// TwinCAT 3 PLC project PLC1
// ProgramVersion: 3.1.4024.12
// libraries:
//   SG_Servo, * (SG)
//   Tc2_Standard, * (Beckhoff Automation GmbH)
//   Tc2_System, * (Beckhoff Automation GmbH)
//   Tc3_Module, * (Beckhoff Automation GmbH)
// project tree:
//   / PlcTask.TcTTO
//   POUs/ MAIN.TcPOU, DeviceState.TcPOU, UN01.TcPOU
// real-time tasks:
//   TASK PlcTask: cycle T#1ms, priority 20, ADS port 350
// motion (NC):
//   TASK NC-Task 1 SAF: cycle T#2ms, priority 4, ADS port 501
//   TASK NC-Task 1 SVB: cycle T#10ms, priority 8, ADS port 511
//   AXIS EM04-M1 (id 1)
//     Dynamic: AccelerationMaximum=2000, DecelerationMaximum=2000, Acceleration=926.842, Deceleration=926.842, Jerk=2000
//     Velo: RefSearch=6.17895, RefSync=6.17895, SlowManual=50, FastManual=200, Fast=617.895, Maximum=200
//     OtherSettings: AllowMotionCmdToSlave=true
//     encoder EncType=19
//       EncPara: ScaleFactorNumerator=12560, ScaleFactorDenominator=1907359744, Inverse=true, MaxCount=#xffffffff
//     drive DrvType=16
//       DrvPara: Inverse=true, MaxCount=#xffffffff, DriveControlDWord=#x00020000
//         Analog: VeloReferenz=679.6845, VeloScale=32, TorqueSetpointScale=10, ScaleFactorActTorque=0.1
//         TimeComp: TaskDelayCycles=1
//     controller CtrType=1
//       CtrPara: PriorControlFactor=1
//         Observer: BandWidth=20
//   AXIS EM05-M1 (id 2)
//     Dynamic: AccelerationMaximum=2000, DecelerationMaximum=2000, Acceleration=926.842, Deceleration=926.842, Jerk=2000
//     Velo: RefSearch=6.17895, RefSync=6.17895, SlowManual=50, FastManual=200, Fast=617.895, Maximum=200
//     OtherSettings: AllowMotionCmdToSlave=true
//     encoder EncType=19
//       EncPara: ScaleFactorNumerator=12560, ScaleFactorDenominator=1907359744, MaxCount=#xffffffff
//     drive DrvType=16
//       DrvPara: MaxCount=#xffffffff, DriveControlDWord=#x00020000
//         Analog: VeloReferenz=679.6845, VeloScale=32, TorqueSetpointScale=10, ScaleFactorActTorque=0.1
//         TimeComp: TaskDelayCycles=1
//     controller CtrType=1
//       CtrPara: PriorControlFactor=1
//         Observer: BandWidth=20
//   AXIS EM07-M1 (id 3)
//     Dynamic: AccelerationMaximum=1000, DecelerationMaximum=1000, Acceleration=2000, Deceleration=2000, Jerk=6000
//     Velo: RefSearch=15.76615, RefSync=15.76615, SlowManual=50, FastManual=250, Fast=1576.615, Maximum=250
//     OtherSettings: AllowMotionCmdToSlave=true
//     encoder EncType=19
//       EncPara: ScaleFactorNumerator=21195, ScaleFactorDenominator=1261436928, Inverse=true, MaxCount=#xffffffff
//     drive DrvType=16
//       DrvPara: Inverse=true, MaxCount=#xffffffff, DriveControlDWord=#x00020000
//         Analog: VeloReferenz=250, VeloScale=32, TorqueSetpointScale=10, ScaleFactorActTorque=0.1
//         TimeComp: TaskDelayCycles=1
//     controller CtrType=1
//       CtrPara: PriorControlFactor=1
//         Observer: BandWidth=20
//   AXIS EM08-M1 (id 4)
//     Dynamic: AccelerationMaximum=1000, DecelerationMaximum=1000, Acceleration=2000, Deceleration=2000, Jerk=6000
//     Velo: RefSearch=15.76615, RefSync=15.76615, SlowManual=50, FastManual=250, Fast=1576.615, Maximum=250
//     OtherSettings: AllowMotionCmdToSlave=true
//     encoder EncType=19
//       EncPara: ScaleFactorNumerator=21195, ScaleFactorDenominator=1261436928, Inverse=true, MaxCount=#xffffffff
//     drive DrvType=16
//       DrvPara: Inverse=true, MaxCount=#xffffffff, DriveControlDWord=#x00020000
//         Analog: VeloReferenz=250, VeloScale=32, TorqueSetpointScale=10, ScaleFactorActTorque=0.1
//         TimeComp: TaskDelayCycles=1
//     controller CtrType=1
//       CtrPara: PriorControlFactor=1
//         Observer: BandWidth=20
// I/O:
//   DEVICE Device 1 (EtherCAT), AmsNetId 5.142.194.67.2.1
//     Term 1 (EK1200) [EK1200-5000 EtherCAT Power supply (2A E-Bus)]
//       Term 2 (EL6631-0010) [EL6631-0010 PROFINET IO Device]
//       Term 3 (EL9011) [EL9011 End Terminal]
//   DEVICE Device 4 (EtherCAT), AmsNetId 5.142.194.67.5.1
//     Term 4 (EK1100) [EK1100 EtherCAT Coupler (2A E-Bus)]
//       Term 5 (EL9576) [EL9576 Brake chopper terminal]
//       Term 6 (EL7221-9014) [EL7221-9014 1Ch. MDP742 Servo motor output stage with OCT (50V, 8A RMS) and STO input]
//         startup 32785:21 := 0E01 // DRV Motor Settings / Commutation offset
//         startup 32785:27 := 01150000 // DRV Motor Settings / Motor speed limitation
//         startup 28688:11 := E803 // DRV Outputs / Torque limitation
//         startup 32784:19 := 5300 // DRV Amplifier Settings / Current loop proportional gain
//         startup 32784:18 := 0500 // DRV Amplifier Settings / Current loop integral time
//         startup 32784:21 := E4000000 // DRV Amplifier Settings / Velocity loop proportional gain
//         startup 32784:20 := 96000000 // DRV Amplifier Settings / Velocity loop integral time
//         startup 32768:1 := 00 // FB Settings / Invert feedback direction
//       Term 7 (EL7221-9014) [EL7221-9014 1Ch. MDP742 Servo motor output stage with OCT (50V, 8A RMS) and STO input]
//         startup 32785:21 := 0E01 // DRV Motor Settings / Commutation offset
//         startup 32785:27 := 01150000 // DRV Motor Settings / Motor speed limitation
//         startup 28688:11 := E803 // DRV Outputs / Torque limitation
//         startup 32784:19 := 5300 // DRV Amplifier Settings / Current loop proportional gain
//         startup 32784:18 := 0500 // DRV Amplifier Settings / Current loop integral time
//         startup 32784:21 := E4000000 // DRV Amplifier Settings / Velocity loop proportional gain
//         startup 32784:20 := 96000000 // DRV Amplifier Settings / Velocity loop integral time
//         startup 32768:1 := 00 // FB Settings / Invert feedback direction
//       Term 8 (EL7221-9014) [EL7221-9014 1Ch. MDP742 Servo motor output stage with OCT (50V, 8A RMS) and STO input]
//         startup 32785:21 := 0E01 // DRV Motor Settings / Commutation offset
//         startup 32785:27 := 01150000 // DRV Motor Settings / Motor speed limitation
//         startup 28688:11 := E803 // DRV Outputs / Torque limitation
//         startup 32784:19 := 5300 // DRV Amplifier Settings / Current loop proportional gain
//         startup 32784:18 := 0500 // DRV Amplifier Settings / Current loop integral time
//         startup 32784:21 := E4000000 // DRV Amplifier Settings / Velocity loop proportional gain
//         startup 32784:20 := 96000000 // DRV Amplifier Settings / Velocity loop integral time
//         startup 32768:1 := 00 // FB Settings / Invert feedback direction
//       Term 9 (EL7221-9014) [EL7221-9014 1Ch. MDP742 Servo motor output stage with OCT (50V, 8A RMS) and STO input]
//         startup 32785:21 := 0E01 // DRV Motor Settings / Commutation offset
//         startup 32785:27 := 01150000 // DRV Motor Settings / Motor speed limitation
//         startup 28688:11 := E803 // DRV Outputs / Torque limitation
//         startup 32784:19 := 5300 // DRV Amplifier Settings / Current loop proportional gain
//         startup 32784:18 := 0500 // DRV Amplifier Settings / Current loop integral time
//         startup 32784:21 := E4000000 // DRV Amplifier Settings / Velocity loop proportional gain
//         startup 32784:20 := 96000000 // DRV Amplifier Settings / Velocity loop integral time
//         startup 32768:1 := 00 // FB Settings / Invert feedback direction
//       Term 7 (EL9011) [EL9011 End Terminal]
//   DEVICE Device 2 (EL6631-0010), AmsNetId 5.109.120.57.3.1
//     el6631-0010 [Beckhoff Automation PROFINET I/O device - EtherCAT slave terminal, V2.33, 2 port diagnostic, MRP and shared device  supported EL6631-0010]
//       modules: Term 1 (DAP Module), Term 2 (Modular)
// variable links:
//   NC-Task 1 SAF/Axes/EM04-M1 <-> Device 4 (EtherCAT)/Term 4 (EK1100)/Term 6 (EL7221-9014)
//     Drive/Inputs/In/nDcOutputTime <-> InfoData/DcOutputShift
//     Drive/Inputs/In/nState1 <-> DRV Statusword/Statusword
//     Drive/Inputs/In/nState2 <-> DRV Statusword/Statusword @bit 8
//     Drive/Inputs/In/nState4 @bit 1 <-> WcState/InputToggle
//     Drive/Inputs/In/nState4 <-> WcState/WcState
//     Drive/Outputs/Out/nCtrl1 <-> DRV Controlword/Controlword
//     Drive/Outputs/Out/nCtrl2 <-> DRV Controlword/Controlword @bit 8
//     Drive/Outputs/Out/nDataOut2 <-> DRV Target velocity/Target velocity
//     Enc/Inputs/In/nDataIn1 <-> FB Position/Position
//     Enc/Inputs/In/nDcInputTime <-> InfoData/DcInputShift
//     Enc/Inputs/In/nState4 @bit 1 <-> WcState/InputToggle
//     Enc/Inputs/In/nState4 <-> WcState/WcState
//   NC-Task 1 SAF/Axes/EM05-M1 <-> Device 4 (EtherCAT)/Term 4 (EK1100)/Term 7 (EL7221-9014)
//     Drive/Inputs/In/nDcOutputTime <-> InfoData/DcOutputShift
//     Drive/Inputs/In/nState1 <-> DRV Statusword/Statusword
//     Drive/Inputs/In/nState2 <-> DRV Statusword/Statusword @bit 8
//     Drive/Inputs/In/nState4 @bit 1 <-> WcState/InputToggle
//     Drive/Inputs/In/nState4 <-> WcState/WcState
//     Drive/Outputs/Out/nCtrl1 <-> DRV Controlword/Controlword
//     Drive/Outputs/Out/nCtrl2 <-> DRV Controlword/Controlword @bit 8
//     Drive/Outputs/Out/nDataOut2 <-> DRV Target velocity/Target velocity
//     Enc/Inputs/In/nDataIn1 <-> FB Position/Position
//     Enc/Inputs/In/nDcInputTime <-> InfoData/DcInputShift
//     Enc/Inputs/In/nState4 @bit 1 <-> WcState/InputToggle
//     Enc/Inputs/In/nState4 <-> WcState/WcState
//   NC-Task 1 SAF/Axes/EM07-M1 <-> Device 4 (EtherCAT)/Term 4 (EK1100)/Term 8 (EL7221-9014)
//     Drive/Inputs/In/nDcOutputTime <-> InfoData/DcOutputShift
//     Drive/Inputs/In/nState1 <-> DRV Statusword/Statusword
//     Drive/Inputs/In/nState2 <-> DRV Statusword/Statusword @bit 8
//     Drive/Inputs/In/nState4 @bit 1 <-> WcState/InputToggle
//     Drive/Inputs/In/nState4 <-> WcState/WcState
//     Drive/Outputs/Out/nCtrl1 <-> DRV Controlword/Controlword
//     Drive/Outputs/Out/nCtrl2 <-> DRV Controlword/Controlword @bit 8
//     Drive/Outputs/Out/nDataOut2 <-> DRV Target velocity/Target velocity
//     Enc/Inputs/In/nDataIn1 <-> FB Position/Position
//     Enc/Inputs/In/nDcInputTime <-> InfoData/DcInputShift
//     Enc/Inputs/In/nState4 @bit 1 <-> WcState/InputToggle
//     Enc/Inputs/In/nState4 <-> WcState/WcState
//   NC-Task 1 SAF/Axes/EM08-M1 <-> Device 4 (EtherCAT)/Term 4 (EK1100)/Term 9 (EL7221-9014)
//     Drive/Inputs/In/nDcOutputTime <-> InfoData/DcOutputShift
//     Drive/Inputs/In/nState1 <-> DRV Statusword/Statusword
//     Drive/Inputs/In/nState2 <-> DRV Statusword/Statusword @bit 8
//     Drive/Inputs/In/nState4 @bit 1 <-> WcState/InputToggle
//     Drive/Inputs/In/nState4 <-> WcState/WcState
//     Drive/Outputs/Out/nCtrl1 <-> DRV Controlword/Controlword
//     Drive/Outputs/Out/nCtrl2 <-> DRV Controlword/Controlword @bit 8
//     Drive/Outputs/Out/nDataOut2 <-> DRV Target velocity/Target velocity
//     Enc/Inputs/In/nDataIn1 <-> FB Position/Position
//     Enc/Inputs/In/nDcInputTime <-> InfoData/DcInputShift
//     Enc/Inputs/In/nState4 @bit 1 <-> WcState/InputToggle
//     Enc/Inputs/In/nState4 <-> WcState/WcState
//   PLC1/PLC1 Instance <-> Device 1 (EtherCAT)
//     PlcTask Inputs/DeviceState.nDev1_DevState <-> Inputs/DevState
//   PLC1/PLC1 Instance <-> Device 1 (EtherCAT)/Term 1 (EK1200)/Term 2 (EL6631-0010)
//     PlcTask Inputs/DeviceState.nProfinetState <-> InfoData/State
//   PLC1/PLC1 Instance <-> Device 2 (EL6631-0010)/el6631-0010
//     PlcTask Inputs/DeviceState.nPnIoBoxState <-> Inputs/PnIoBoxState
//     PlcTask Inputs/UN01.inf_EM04_M1.in/data <-> API/Term 2 (Modular)/EM04-M1/Inputs/1 Byte Output[0]
//     PlcTask Inputs/UN01.inf_EM05_M1.in/data <-> API/Term 2 (Modular)/EM05-M1/Inputs/1 Byte Output[0]
//     PlcTask Inputs/UN01.inf_EM07_M1.in/data <-> API/Term 2 (Modular)/EM07-M1/Inputs/1 Byte Output[0]
//     PlcTask Inputs/UN01.inf_EM08_M1.in/data <-> API/Term 2 (Modular)/EM08-M1/Inputs/1 Byte Output[0]
//     PlcTask Inputs/UN01.inf_EM04_M1.in/data @bit 80 <-> API/Term 2 (Modular)/EM04-M1/Inputs/1 Byte Output[10]
//     PlcTask Inputs/UN01.inf_EM04_M1.in/data @bit 88 <-> API/Term 2 (Modular)/EM04-M1/Inputs/1 Byte Output[11]
//     PlcTask Inputs/UN01.inf_EM04_M1.in/data @bit 96 <-> API/Term 2 (Modular)/EM04-M1/Inputs/1 Byte Output[12]
//     PlcTask Inputs/UN01.inf_EM04_M1.in/data @bit 104 <-> API/Term 2 (Modular)/EM04-M1/Inputs/1 Byte Output[13]
//     PlcTask Inputs/UN01.inf_EM04_M1.in/data @bit 112 <-> API/Term 2 (Modular)/EM04-M1/Inputs/1 Byte Output[14]
//     PlcTask Inputs/UN01.inf_EM04_M1.in/data @bit 120 <-> API/Term 2 (Modular)/EM04-M1/Inputs/1 Byte Output[15]
//     PlcTask Inputs/UN01.inf_EM04_M1.in/data @bit 128 <-> API/Term 2 (Modular)/EM04-M1/Inputs/1 Byte Output[16]
//     PlcTask Inputs/UN01.inf_EM04_M1.in/data @bit 136 <-> API/Term 2 (Modular)/EM04-M1/Inputs/1 Byte Output[17]
//     PlcTask Inputs/UN01.inf_EM04_M1.in/data @bit 144 <-> API/Term 2 (Modular)/EM04-M1/Inputs/1 Byte Output[18]
//     PlcTask Inputs/UN01.inf_EM04_M1.in/data @bit 152 <-> API/Term 2 (Modular)/EM04-M1/Inputs/1 Byte Output[19]
//     PlcTask Inputs/UN01.inf_EM04_M1.in/data @bit 8 <-> API/Term 2 (Modular)/EM04-M1/Inputs/1 Byte Output[1]
//     PlcTask Inputs/UN01.inf_EM04_M1.in/data @bit 160 <-> API/Term 2 (Modular)/EM04-M1/Inputs/1 Byte Output[20]
//     PlcTask Inputs/UN01.inf_EM04_M1.in/data @bit 168 <-> API/Term 2 (Modular)/EM04-M1/Inputs/1 Byte Output[21]
//     PlcTask Inputs/UN01.inf_EM04_M1.in/data @bit 176 <-> API/Term 2 (Modular)/EM04-M1/Inputs/1 Byte Output[22]
//     PlcTask Inputs/UN01.inf_EM04_M1.in/data @bit 184 <-> API/Term 2 (Modular)/EM04-M1/Inputs/1 Byte Output[23]
//     PlcTask Inputs/UN01.inf_EM04_M1.in/data @bit 192 <-> API/Term 2 (Modular)/EM04-M1/Inputs/1 Byte Output[24]
//     PlcTask Inputs/UN01.inf_EM04_M1.in/data @bit 200 <-> API/Term 2 (Modular)/EM04-M1/Inputs/1 Byte Output[25]
//     PlcTask Inputs/UN01.inf_EM04_M1.in/data @bit 208 <-> API/Term 2 (Modular)/EM04-M1/Inputs/1 Byte Output[26]
//     PlcTask Inputs/UN01.inf_EM04_M1.in/data @bit 216 <-> API/Term 2 (Modular)/EM04-M1/Inputs/1 Byte Output[27]
//     PlcTask Inputs/UN01.inf_EM04_M1.in/data @bit 224 <-> API/Term 2 (Modular)/EM04-M1/Inputs/1 Byte Output[28]
//     PlcTask Inputs/UN01.inf_EM04_M1.in/data @bit 232 <-> API/Term 2 (Modular)/EM04-M1/Inputs/1 Byte Output[29]
//     PlcTask Inputs/UN01.inf_EM04_M1.in/data @bit 16 <-> API/Term 2 (Modular)/EM04-M1/Inputs/1 Byte Output[2]
//     PlcTask Inputs/UN01.inf_EM04_M1.in/data @bit 240 <-> API/Term 2 (Modular)/EM04-M1/Inputs/1 Byte Output[30]
//     PlcTask Inputs/UN01.inf_EM04_M1.in/data @bit 248 <-> API/Term 2 (Modular)/EM04-M1/Inputs/1 Byte Output[31]
//     PlcTask Inputs/UN01.inf_EM04_M1.in/data @bit 24 <-> API/Term 2 (Modular)/EM04-M1/Inputs/1 Byte Output[3]
//     PlcTask Inputs/UN01.inf_EM04_M1.in/data @bit 32 <-> API/Term 2 (Modular)/EM04-M1/Inputs/1 Byte Output[4]
//     PlcTask Inputs/UN01.inf_EM04_M1.in/data @bit 40 <-> API/Term 2 (Modular)/EM04-M1/Inputs/1 Byte Output[5]
//     PlcTask Inputs/UN01.inf_EM04_M1.in/data @bit 48 <-> API/Term 2 (Modular)/EM04-M1/Inputs/1 Byte Output[6]
//     PlcTask Inputs/UN01.inf_EM04_M1.in/data @bit 56 <-> API/Term 2 (Modular)/EM04-M1/Inputs/1 Byte Output[7]
//     PlcTask Inputs/UN01.inf_EM04_M1.in/data @bit 64 <-> API/Term 2 (Modular)/EM04-M1/Inputs/1 Byte Output[8]
//     PlcTask Inputs/UN01.inf_EM04_M1.in/data @bit 72 <-> API/Term 2 (Modular)/EM04-M1/Inputs/1 Byte Output[9]
//     PlcTask Inputs/UN01.inf_EM05_M1.in/data @bit 80 <-> API/Term 2 (Modular)/EM05-M1/Inputs/1 Byte Output[10]
//     PlcTask Inputs/UN01.inf_EM05_M1.in/data @bit 88 <-> API/Term 2 (Modular)/EM05-M1/Inputs/1 Byte Output[11]
//     PlcTask Inputs/UN01.inf_EM05_M1.in/data @bit 96 <-> API/Term 2 (Modular)/EM05-M1/Inputs/1 Byte Output[12]
//     PlcTask Inputs/UN01.inf_EM05_M1.in/data @bit 104 <-> API/Term 2 (Modular)/EM05-M1/Inputs/1 Byte Output[13]
//     PlcTask Inputs/UN01.inf_EM05_M1.in/data @bit 112 <-> API/Term 2 (Modular)/EM05-M1/Inputs/1 Byte Output[14]
//     PlcTask Inputs/UN01.inf_EM05_M1.in/data @bit 120 <-> API/Term 2 (Modular)/EM05-M1/Inputs/1 Byte Output[15]
//     PlcTask Inputs/UN01.inf_EM05_M1.in/data @bit 128 <-> API/Term 2 (Modular)/EM05-M1/Inputs/1 Byte Output[16]
//     PlcTask Inputs/UN01.inf_EM05_M1.in/data @bit 136 <-> API/Term 2 (Modular)/EM05-M1/Inputs/1 Byte Output[17]
//     PlcTask Inputs/UN01.inf_EM05_M1.in/data @bit 144 <-> API/Term 2 (Modular)/EM05-M1/Inputs/1 Byte Output[18]
//     PlcTask Inputs/UN01.inf_EM05_M1.in/data @bit 152 <-> API/Term 2 (Modular)/EM05-M1/Inputs/1 Byte Output[19]
//     PlcTask Inputs/UN01.inf_EM05_M1.in/data @bit 8 <-> API/Term 2 (Modular)/EM05-M1/Inputs/1 Byte Output[1]
//     PlcTask Inputs/UN01.inf_EM05_M1.in/data @bit 160 <-> API/Term 2 (Modular)/EM05-M1/Inputs/1 Byte Output[20]
//     PlcTask Inputs/UN01.inf_EM05_M1.in/data @bit 168 <-> API/Term 2 (Modular)/EM05-M1/Inputs/1 Byte Output[21]
//     PlcTask Inputs/UN01.inf_EM05_M1.in/data @bit 176 <-> API/Term 2 (Modular)/EM05-M1/Inputs/1 Byte Output[22]
//     PlcTask Inputs/UN01.inf_EM05_M1.in/data @bit 184 <-> API/Term 2 (Modular)/EM05-M1/Inputs/1 Byte Output[23]
//     PlcTask Inputs/UN01.inf_EM05_M1.in/data @bit 192 <-> API/Term 2 (Modular)/EM05-M1/Inputs/1 Byte Output[24]
//     PlcTask Inputs/UN01.inf_EM05_M1.in/data @bit 200 <-> API/Term 2 (Modular)/EM05-M1/Inputs/1 Byte Output[25]
//     PlcTask Inputs/UN01.inf_EM05_M1.in/data @bit 208 <-> API/Term 2 (Modular)/EM05-M1/Inputs/1 Byte Output[26]
//     PlcTask Inputs/UN01.inf_EM05_M1.in/data @bit 216 <-> API/Term 2 (Modular)/EM05-M1/Inputs/1 Byte Output[27]
//     PlcTask Inputs/UN01.inf_EM05_M1.in/data @bit 224 <-> API/Term 2 (Modular)/EM05-M1/Inputs/1 Byte Output[28]
//     PlcTask Inputs/UN01.inf_EM05_M1.in/data @bit 232 <-> API/Term 2 (Modular)/EM05-M1/Inputs/1 Byte Output[29]
//     PlcTask Inputs/UN01.inf_EM05_M1.in/data @bit 16 <-> API/Term 2 (Modular)/EM05-M1/Inputs/1 Byte Output[2]
//     PlcTask Inputs/UN01.inf_EM05_M1.in/data @bit 240 <-> API/Term 2 (Modular)/EM05-M1/Inputs/1 Byte Output[30]
//     PlcTask Inputs/UN01.inf_EM05_M1.in/data @bit 248 <-> API/Term 2 (Modular)/EM05-M1/Inputs/1 Byte Output[31]
//     PlcTask Inputs/UN01.inf_EM05_M1.in/data @bit 24 <-> API/Term 2 (Modular)/EM05-M1/Inputs/1 Byte Output[3]
//     PlcTask Inputs/UN01.inf_EM05_M1.in/data @bit 32 <-> API/Term 2 (Modular)/EM05-M1/Inputs/1 Byte Output[4]
//     PlcTask Inputs/UN01.inf_EM05_M1.in/data @bit 40 <-> API/Term 2 (Modular)/EM05-M1/Inputs/1 Byte Output[5]
//     PlcTask Inputs/UN01.inf_EM05_M1.in/data @bit 48 <-> API/Term 2 (Modular)/EM05-M1/Inputs/1 Byte Output[6]
//     PlcTask Inputs/UN01.inf_EM05_M1.in/data @bit 56 <-> API/Term 2 (Modular)/EM05-M1/Inputs/1 Byte Output[7]
//     PlcTask Inputs/UN01.inf_EM05_M1.in/data @bit 64 <-> API/Term 2 (Modular)/EM05-M1/Inputs/1 Byte Output[8]
//     PlcTask Inputs/UN01.inf_EM05_M1.in/data @bit 72 <-> API/Term 2 (Modular)/EM05-M1/Inputs/1 Byte Output[9]
//     PlcTask Inputs/UN01.inf_EM07_M1.in/data @bit 80 <-> API/Term 2 (Modular)/EM07-M1/Inputs/1 Byte Output[10]
//     PlcTask Inputs/UN01.inf_EM07_M1.in/data @bit 88 <-> API/Term 2 (Modular)/EM07-M1/Inputs/1 Byte Output[11]
//     PlcTask Inputs/UN01.inf_EM07_M1.in/data @bit 96 <-> API/Term 2 (Modular)/EM07-M1/Inputs/1 Byte Output[12]
//     PlcTask Inputs/UN01.inf_EM07_M1.in/data @bit 104 <-> API/Term 2 (Modular)/EM07-M1/Inputs/1 Byte Output[13]
//     PlcTask Inputs/UN01.inf_EM07_M1.in/data @bit 112 <-> API/Term 2 (Modular)/EM07-M1/Inputs/1 Byte Output[14]
//     PlcTask Inputs/UN01.inf_EM07_M1.in/data @bit 120 <-> API/Term 2 (Modular)/EM07-M1/Inputs/1 Byte Output[15]
//     PlcTask Inputs/UN01.inf_EM07_M1.in/data @bit 128 <-> API/Term 2 (Modular)/EM07-M1/Inputs/1 Byte Output[16]
//     PlcTask Inputs/UN01.inf_EM07_M1.in/data @bit 136 <-> API/Term 2 (Modular)/EM07-M1/Inputs/1 Byte Output[17]
//     PlcTask Inputs/UN01.inf_EM07_M1.in/data @bit 144 <-> API/Term 2 (Modular)/EM07-M1/Inputs/1 Byte Output[18]
//     PlcTask Inputs/UN01.inf_EM07_M1.in/data @bit 152 <-> API/Term 2 (Modular)/EM07-M1/Inputs/1 Byte Output[19]
//     PlcTask Inputs/UN01.inf_EM07_M1.in/data @bit 8 <-> API/Term 2 (Modular)/EM07-M1/Inputs/1 Byte Output[1]
//     PlcTask Inputs/UN01.inf_EM07_M1.in/data @bit 160 <-> API/Term 2 (Modular)/EM07-M1/Inputs/1 Byte Output[20]
//     PlcTask Inputs/UN01.inf_EM07_M1.in/data @bit 168 <-> API/Term 2 (Modular)/EM07-M1/Inputs/1 Byte Output[21]
//     PlcTask Inputs/UN01.inf_EM07_M1.in/data @bit 176 <-> API/Term 2 (Modular)/EM07-M1/Inputs/1 Byte Output[22]
//     PlcTask Inputs/UN01.inf_EM07_M1.in/data @bit 184 <-> API/Term 2 (Modular)/EM07-M1/Inputs/1 Byte Output[23]
//     PlcTask Inputs/UN01.inf_EM07_M1.in/data @bit 192 <-> API/Term 2 (Modular)/EM07-M1/Inputs/1 Byte Output[24]
//     PlcTask Inputs/UN01.inf_EM07_M1.in/data @bit 200 <-> API/Term 2 (Modular)/EM07-M1/Inputs/1 Byte Output[25]
//     PlcTask Inputs/UN01.inf_EM07_M1.in/data @bit 208 <-> API/Term 2 (Modular)/EM07-M1/Inputs/1 Byte Output[26]
//     PlcTask Inputs/UN01.inf_EM07_M1.in/data @bit 216 <-> API/Term 2 (Modular)/EM07-M1/Inputs/1 Byte Output[27]
//     PlcTask Inputs/UN01.inf_EM07_M1.in/data @bit 224 <-> API/Term 2 (Modular)/EM07-M1/Inputs/1 Byte Output[28]
//     PlcTask Inputs/UN01.inf_EM07_M1.in/data @bit 232 <-> API/Term 2 (Modular)/EM07-M1/Inputs/1 Byte Output[29]
//     PlcTask Inputs/UN01.inf_EM07_M1.in/data @bit 16 <-> API/Term 2 (Modular)/EM07-M1/Inputs/1 Byte Output[2]
//     PlcTask Inputs/UN01.inf_EM07_M1.in/data @bit 240 <-> API/Term 2 (Modular)/EM07-M1/Inputs/1 Byte Output[30]
//     PlcTask Inputs/UN01.inf_EM07_M1.in/data @bit 248 <-> API/Term 2 (Modular)/EM07-M1/Inputs/1 Byte Output[31]
//     PlcTask Inputs/UN01.inf_EM07_M1.in/data @bit 24 <-> API/Term 2 (Modular)/EM07-M1/Inputs/1 Byte Output[3]
//     PlcTask Inputs/UN01.inf_EM07_M1.in/data @bit 32 <-> API/Term 2 (Modular)/EM07-M1/Inputs/1 Byte Output[4]
//     PlcTask Inputs/UN01.inf_EM07_M1.in/data @bit 40 <-> API/Term 2 (Modular)/EM07-M1/Inputs/1 Byte Output[5]
//     PlcTask Inputs/UN01.inf_EM07_M1.in/data @bit 48 <-> API/Term 2 (Modular)/EM07-M1/Inputs/1 Byte Output[6]
//     PlcTask Inputs/UN01.inf_EM07_M1.in/data @bit 56 <-> API/Term 2 (Modular)/EM07-M1/Inputs/1 Byte Output[7]
//     PlcTask Inputs/UN01.inf_EM07_M1.in/data @bit 64 <-> API/Term 2 (Modular)/EM07-M1/Inputs/1 Byte Output[8]
//     PlcTask Inputs/UN01.inf_EM07_M1.in/data @bit 72 <-> API/Term 2 (Modular)/EM07-M1/Inputs/1 Byte Output[9]
//     PlcTask Inputs/UN01.inf_EM08_M1.in/data @bit 80 <-> API/Term 2 (Modular)/EM08-M1/Inputs/1 Byte Output[10]
//     PlcTask Inputs/UN01.inf_EM08_M1.in/data @bit 88 <-> API/Term 2 (Modular)/EM08-M1/Inputs/1 Byte Output[11]
//     PlcTask Inputs/UN01.inf_EM08_M1.in/data @bit 96 <-> API/Term 2 (Modular)/EM08-M1/Inputs/1 Byte Output[12]
//     PlcTask Inputs/UN01.inf_EM08_M1.in/data @bit 104 <-> API/Term 2 (Modular)/EM08-M1/Inputs/1 Byte Output[13]
//     PlcTask Inputs/UN01.inf_EM08_M1.in/data @bit 112 <-> API/Term 2 (Modular)/EM08-M1/Inputs/1 Byte Output[14]
//     PlcTask Inputs/UN01.inf_EM08_M1.in/data @bit 120 <-> API/Term 2 (Modular)/EM08-M1/Inputs/1 Byte Output[15]
//     PlcTask Inputs/UN01.inf_EM08_M1.in/data @bit 128 <-> API/Term 2 (Modular)/EM08-M1/Inputs/1 Byte Output[16]
//     PlcTask Inputs/UN01.inf_EM08_M1.in/data @bit 136 <-> API/Term 2 (Modular)/EM08-M1/Inputs/1 Byte Output[17]
//     PlcTask Inputs/UN01.inf_EM08_M1.in/data @bit 144 <-> API/Term 2 (Modular)/EM08-M1/Inputs/1 Byte Output[18]
//     PlcTask Inputs/UN01.inf_EM08_M1.in/data @bit 152 <-> API/Term 2 (Modular)/EM08-M1/Inputs/1 Byte Output[19]
//     PlcTask Inputs/UN01.inf_EM08_M1.in/data @bit 8 <-> API/Term 2 (Modular)/EM08-M1/Inputs/1 Byte Output[1]
//     PlcTask Inputs/UN01.inf_EM08_M1.in/data @bit 160 <-> API/Term 2 (Modular)/EM08-M1/Inputs/1 Byte Output[20]
//     PlcTask Inputs/UN01.inf_EM08_M1.in/data @bit 168 <-> API/Term 2 (Modular)/EM08-M1/Inputs/1 Byte Output[21]
//     PlcTask Inputs/UN01.inf_EM08_M1.in/data @bit 176 <-> API/Term 2 (Modular)/EM08-M1/Inputs/1 Byte Output[22]
//     PlcTask Inputs/UN01.inf_EM08_M1.in/data @bit 184 <-> API/Term 2 (Modular)/EM08-M1/Inputs/1 Byte Output[23]
//     PlcTask Inputs/UN01.inf_EM08_M1.in/data @bit 192 <-> API/Term 2 (Modular)/EM08-M1/Inputs/1 Byte Output[24]
//     PlcTask Inputs/UN01.inf_EM08_M1.in/data @bit 200 <-> API/Term 2 (Modular)/EM08-M1/Inputs/1 Byte Output[25]
//     PlcTask Inputs/UN01.inf_EM08_M1.in/data @bit 208 <-> API/Term 2 (Modular)/EM08-M1/Inputs/1 Byte Output[26]
//     PlcTask Inputs/UN01.inf_EM08_M1.in/data @bit 216 <-> API/Term 2 (Modular)/EM08-M1/Inputs/1 Byte Output[27]
//     PlcTask Inputs/UN01.inf_EM08_M1.in/data @bit 224 <-> API/Term 2 (Modular)/EM08-M1/Inputs/1 Byte Output[28]
//     PlcTask Inputs/UN01.inf_EM08_M1.in/data @bit 232 <-> API/Term 2 (Modular)/EM08-M1/Inputs/1 Byte Output[29]
//     PlcTask Inputs/UN01.inf_EM08_M1.in/data @bit 16 <-> API/Term 2 (Modular)/EM08-M1/Inputs/1 Byte Output[2]
//     PlcTask Inputs/UN01.inf_EM08_M1.in/data @bit 240 <-> API/Term 2 (Modular)/EM08-M1/Inputs/1 Byte Output[30]
//     PlcTask Inputs/UN01.inf_EM08_M1.in/data @bit 248 <-> API/Term 2 (Modular)/EM08-M1/Inputs/1 Byte Output[31]
//     PlcTask Inputs/UN01.inf_EM08_M1.in/data @bit 24 <-> API/Term 2 (Modular)/EM08-M1/Inputs/1 Byte Output[3]
//     PlcTask Inputs/UN01.inf_EM08_M1.in/data @bit 32 <-> API/Term 2 (Modular)/EM08-M1/Inputs/1 Byte Output[4]
//     PlcTask Inputs/UN01.inf_EM08_M1.in/data @bit 40 <-> API/Term 2 (Modular)/EM08-M1/Inputs/1 Byte Output[5]
//     PlcTask Inputs/UN01.inf_EM08_M1.in/data @bit 48 <-> API/Term 2 (Modular)/EM08-M1/Inputs/1 Byte Output[6]
//     PlcTask Inputs/UN01.inf_EM08_M1.in/data @bit 56 <-> API/Term 2 (Modular)/EM08-M1/Inputs/1 Byte Output[7]
//     PlcTask Inputs/UN01.inf_EM08_M1.in/data @bit 64 <-> API/Term 2 (Modular)/EM08-M1/Inputs/1 Byte Output[8]
//     PlcTask Inputs/UN01.inf_EM08_M1.in/data @bit 72 <-> API/Term 2 (Modular)/EM08-M1/Inputs/1 Byte Output[9]
//     PlcTask Outputs/DeviceState.nPnIoBoxCtrl <-> Outputs/PnIoBoxCtrl
//     PlcTask Outputs/UN01.inf_EM04_M1.out/data <-> API/Term 2 (Modular)/EM04-M1/Outputs/1 Byte Input[0]
//     PlcTask Outputs/UN01.inf_EM05_M1.out/data <-> API/Term 2 (Modular)/EM05-M1/Outputs/1 Byte Input[0]
//     PlcTask Outputs/UN01.inf_EM07_M1.out/data <-> API/Term 2 (Modular)/EM07-M1/Outputs/1 Byte Input[0]
//     PlcTask Outputs/UN01.inf_EM08_M1.out/data <-> API/Term 2 (Modular)/EM08-M1/Outputs/1 Byte Input[0]
//     PlcTask Outputs/UN01.inf_EM04_M1.out/data @bit 80 <-> API/Term 2 (Modular)/EM04-M1/Outputs/1 Byte Input[10]
//     PlcTask Outputs/UN01.inf_EM04_M1.out/data @bit 88 <-> API/Term 2 (Modular)/EM04-M1/Outputs/1 Byte Input[11]
//     PlcTask Outputs/UN01.inf_EM04_M1.out/data @bit 96 <-> API/Term 2 (Modular)/EM04-M1/Outputs/1 Byte Input[12]
//     PlcTask Outputs/UN01.inf_EM04_M1.out/data @bit 104 <-> API/Term 2 (Modular)/EM04-M1/Outputs/1 Byte Input[13]
//     PlcTask Outputs/UN01.inf_EM04_M1.out/data @bit 112 <-> API/Term 2 (Modular)/EM04-M1/Outputs/1 Byte Input[14]
//     PlcTask Outputs/UN01.inf_EM04_M1.out/data @bit 120 <-> API/Term 2 (Modular)/EM04-M1/Outputs/1 Byte Input[15]
//     PlcTask Outputs/UN01.inf_EM04_M1.out/data @bit 128 <-> API/Term 2 (Modular)/EM04-M1/Outputs/1 Byte Input[16]
//     PlcTask Outputs/UN01.inf_EM04_M1.out/data @bit 136 <-> API/Term 2 (Modular)/EM04-M1/Outputs/1 Byte Input[17]
//     PlcTask Outputs/UN01.inf_EM04_M1.out/data @bit 144 <-> API/Term 2 (Modular)/EM04-M1/Outputs/1 Byte Input[18]
//     PlcTask Outputs/UN01.inf_EM04_M1.out/data @bit 152 <-> API/Term 2 (Modular)/EM04-M1/Outputs/1 Byte Input[19]
//     PlcTask Outputs/UN01.inf_EM04_M1.out/data @bit 8 <-> API/Term 2 (Modular)/EM04-M1/Outputs/1 Byte Input[1]
//     PlcTask Outputs/UN01.inf_EM04_M1.out/data @bit 160 <-> API/Term 2 (Modular)/EM04-M1/Outputs/1 Byte Input[20]
//     PlcTask Outputs/UN01.inf_EM04_M1.out/data @bit 168 <-> API/Term 2 (Modular)/EM04-M1/Outputs/1 Byte Input[21]
//     PlcTask Outputs/UN01.inf_EM04_M1.out/data @bit 176 <-> API/Term 2 (Modular)/EM04-M1/Outputs/1 Byte Input[22]
//     PlcTask Outputs/UN01.inf_EM04_M1.out/data @bit 184 <-> API/Term 2 (Modular)/EM04-M1/Outputs/1 Byte Input[23]
//     PlcTask Outputs/UN01.inf_EM04_M1.out/data @bit 192 <-> API/Term 2 (Modular)/EM04-M1/Outputs/1 Byte Input[24]
//     PlcTask Outputs/UN01.inf_EM04_M1.out/data @bit 200 <-> API/Term 2 (Modular)/EM04-M1/Outputs/1 Byte Input[25]
//     PlcTask Outputs/UN01.inf_EM04_M1.out/data @bit 208 <-> API/Term 2 (Modular)/EM04-M1/Outputs/1 Byte Input[26]
//     PlcTask Outputs/UN01.inf_EM04_M1.out/data @bit 216 <-> API/Term 2 (Modular)/EM04-M1/Outputs/1 Byte Input[27]
//     PlcTask Outputs/UN01.inf_EM04_M1.out/data @bit 224 <-> API/Term 2 (Modular)/EM04-M1/Outputs/1 Byte Input[28]
//     PlcTask Outputs/UN01.inf_EM04_M1.out/data @bit 232 <-> API/Term 2 (Modular)/EM04-M1/Outputs/1 Byte Input[29]
//     PlcTask Outputs/UN01.inf_EM04_M1.out/data @bit 16 <-> API/Term 2 (Modular)/EM04-M1/Outputs/1 Byte Input[2]
//     PlcTask Outputs/UN01.inf_EM04_M1.out/data @bit 240 <-> API/Term 2 (Modular)/EM04-M1/Outputs/1 Byte Input[30]
//     PlcTask Outputs/UN01.inf_EM04_M1.out/data @bit 248 <-> API/Term 2 (Modular)/EM04-M1/Outputs/1 Byte Input[31]
//     PlcTask Outputs/UN01.inf_EM04_M1.out/data @bit 24 <-> API/Term 2 (Modular)/EM04-M1/Outputs/1 Byte Input[3]
//     PlcTask Outputs/UN01.inf_EM04_M1.out/data @bit 32 <-> API/Term 2 (Modular)/EM04-M1/Outputs/1 Byte Input[4]
//     PlcTask Outputs/UN01.inf_EM04_M1.out/data @bit 40 <-> API/Term 2 (Modular)/EM04-M1/Outputs/1 Byte Input[5]
//     PlcTask Outputs/UN01.inf_EM04_M1.out/data @bit 48 <-> API/Term 2 (Modular)/EM04-M1/Outputs/1 Byte Input[6]
//     PlcTask Outputs/UN01.inf_EM04_M1.out/data @bit 56 <-> API/Term 2 (Modular)/EM04-M1/Outputs/1 Byte Input[7]
//     PlcTask Outputs/UN01.inf_EM04_M1.out/data @bit 64 <-> API/Term 2 (Modular)/EM04-M1/Outputs/1 Byte Input[8]
//     PlcTask Outputs/UN01.inf_EM04_M1.out/data @bit 72 <-> API/Term 2 (Modular)/EM04-M1/Outputs/1 Byte Input[9]
//     PlcTask Outputs/UN01.inf_EM05_M1.out/data @bit 80 <-> API/Term 2 (Modular)/EM05-M1/Outputs/1 Byte Input[10]
//     PlcTask Outputs/UN01.inf_EM05_M1.out/data @bit 88 <-> API/Term 2 (Modular)/EM05-M1/Outputs/1 Byte Input[11]
//     PlcTask Outputs/UN01.inf_EM05_M1.out/data @bit 96 <-> API/Term 2 (Modular)/EM05-M1/Outputs/1 Byte Input[12]
//     PlcTask Outputs/UN01.inf_EM05_M1.out/data @bit 104 <-> API/Term 2 (Modular)/EM05-M1/Outputs/1 Byte Input[13]
//     PlcTask Outputs/UN01.inf_EM05_M1.out/data @bit 112 <-> API/Term 2 (Modular)/EM05-M1/Outputs/1 Byte Input[14]
//     PlcTask Outputs/UN01.inf_EM05_M1.out/data @bit 120 <-> API/Term 2 (Modular)/EM05-M1/Outputs/1 Byte Input[15]
//     PlcTask Outputs/UN01.inf_EM05_M1.out/data @bit 128 <-> API/Term 2 (Modular)/EM05-M1/Outputs/1 Byte Input[16]
//     PlcTask Outputs/UN01.inf_EM05_M1.out/data @bit 136 <-> API/Term 2 (Modular)/EM05-M1/Outputs/1 Byte Input[17]
//     PlcTask Outputs/UN01.inf_EM05_M1.out/data @bit 144 <-> API/Term 2 (Modular)/EM05-M1/Outputs/1 Byte Input[18]
//     PlcTask Outputs/UN01.inf_EM05_M1.out/data @bit 152 <-> API/Term 2 (Modular)/EM05-M1/Outputs/1 Byte Input[19]
//     PlcTask Outputs/UN01.inf_EM05_M1.out/data @bit 8 <-> API/Term 2 (Modular)/EM05-M1/Outputs/1 Byte Input[1]
//     PlcTask Outputs/UN01.inf_EM05_M1.out/data @bit 160 <-> API/Term 2 (Modular)/EM05-M1/Outputs/1 Byte Input[20]
//     PlcTask Outputs/UN01.inf_EM05_M1.out/data @bit 168 <-> API/Term 2 (Modular)/EM05-M1/Outputs/1 Byte Input[21]
//     PlcTask Outputs/UN01.inf_EM05_M1.out/data @bit 176 <-> API/Term 2 (Modular)/EM05-M1/Outputs/1 Byte Input[22]
//     PlcTask Outputs/UN01.inf_EM05_M1.out/data @bit 184 <-> API/Term 2 (Modular)/EM05-M1/Outputs/1 Byte Input[23]
//     PlcTask Outputs/UN01.inf_EM05_M1.out/data @bit 192 <-> API/Term 2 (Modular)/EM05-M1/Outputs/1 Byte Input[24]
//     PlcTask Outputs/UN01.inf_EM05_M1.out/data @bit 200 <-> API/Term 2 (Modular)/EM05-M1/Outputs/1 Byte Input[25]
//     PlcTask Outputs/UN01.inf_EM05_M1.out/data @bit 208 <-> API/Term 2 (Modular)/EM05-M1/Outputs/1 Byte Input[26]
//     PlcTask Outputs/UN01.inf_EM05_M1.out/data @bit 216 <-> API/Term 2 (Modular)/EM05-M1/Outputs/1 Byte Input[27]
//     PlcTask Outputs/UN01.inf_EM05_M1.out/data @bit 224 <-> API/Term 2 (Modular)/EM05-M1/Outputs/1 Byte Input[28]
//     PlcTask Outputs/UN01.inf_EM05_M1.out/data @bit 232 <-> API/Term 2 (Modular)/EM05-M1/Outputs/1 Byte Input[29]
//     PlcTask Outputs/UN01.inf_EM05_M1.out/data @bit 16 <-> API/Term 2 (Modular)/EM05-M1/Outputs/1 Byte Input[2]
//     PlcTask Outputs/UN01.inf_EM05_M1.out/data @bit 240 <-> API/Term 2 (Modular)/EM05-M1/Outputs/1 Byte Input[30]
//     PlcTask Outputs/UN01.inf_EM05_M1.out/data @bit 248 <-> API/Term 2 (Modular)/EM05-M1/Outputs/1 Byte Input[31]
//     PlcTask Outputs/UN01.inf_EM05_M1.out/data @bit 24 <-> API/Term 2 (Modular)/EM05-M1/Outputs/1 Byte Input[3]
//     PlcTask Outputs/UN01.inf_EM05_M1.out/data @bit 32 <-> API/Term 2 (Modular)/EM05-M1/Outputs/1 Byte Input[4]
//     PlcTask Outputs/UN01.inf_EM05_M1.out/data @bit 40 <-> API/Term 2 (Modular)/EM05-M1/Outputs/1 Byte Input[5]
//     PlcTask Outputs/UN01.inf_EM05_M1.out/data @bit 48 <-> API/Term 2 (Modular)/EM05-M1/Outputs/1 Byte Input[6]
//     PlcTask Outputs/UN01.inf_EM05_M1.out/data @bit 56 <-> API/Term 2 (Modular)/EM05-M1/Outputs/1 Byte Input[7]
//     PlcTask Outputs/UN01.inf_EM05_M1.out/data @bit 64 <-> API/Term 2 (Modular)/EM05-M1/Outputs/1 Byte Input[8]
//     PlcTask Outputs/UN01.inf_EM05_M1.out/data @bit 72 <-> API/Term 2 (Modular)/EM05-M1/Outputs/1 Byte Input[9]
//     PlcTask Outputs/UN01.inf_EM07_M1.out/data @bit 80 <-> API/Term 2 (Modular)/EM07-M1/Outputs/1 Byte Input[10]
//     PlcTask Outputs/UN01.inf_EM07_M1.out/data @bit 88 <-> API/Term 2 (Modular)/EM07-M1/Outputs/1 Byte Input[11]
//     PlcTask Outputs/UN01.inf_EM07_M1.out/data @bit 96 <-> API/Term 2 (Modular)/EM07-M1/Outputs/1 Byte Input[12]
//     PlcTask Outputs/UN01.inf_EM07_M1.out/data @bit 104 <-> API/Term 2 (Modular)/EM07-M1/Outputs/1 Byte Input[13]
//     PlcTask Outputs/UN01.inf_EM07_M1.out/data @bit 112 <-> API/Term 2 (Modular)/EM07-M1/Outputs/1 Byte Input[14]
//     PlcTask Outputs/UN01.inf_EM07_M1.out/data @bit 120 <-> API/Term 2 (Modular)/EM07-M1/Outputs/1 Byte Input[15]
//     PlcTask Outputs/UN01.inf_EM07_M1.out/data @bit 128 <-> API/Term 2 (Modular)/EM07-M1/Outputs/1 Byte Input[16]
//     PlcTask Outputs/UN01.inf_EM07_M1.out/data @bit 136 <-> API/Term 2 (Modular)/EM07-M1/Outputs/1 Byte Input[17]
//     PlcTask Outputs/UN01.inf_EM07_M1.out/data @bit 144 <-> API/Term 2 (Modular)/EM07-M1/Outputs/1 Byte Input[18]
//     PlcTask Outputs/UN01.inf_EM07_M1.out/data @bit 152 <-> API/Term 2 (Modular)/EM07-M1/Outputs/1 Byte Input[19]
//     PlcTask Outputs/UN01.inf_EM07_M1.out/data @bit 8 <-> API/Term 2 (Modular)/EM07-M1/Outputs/1 Byte Input[1]
//     PlcTask Outputs/UN01.inf_EM07_M1.out/data @bit 160 <-> API/Term 2 (Modular)/EM07-M1/Outputs/1 Byte Input[20]
//     PlcTask Outputs/UN01.inf_EM07_M1.out/data @bit 168 <-> API/Term 2 (Modular)/EM07-M1/Outputs/1 Byte Input[21]
//     PlcTask Outputs/UN01.inf_EM07_M1.out/data @bit 176 <-> API/Term 2 (Modular)/EM07-M1/Outputs/1 Byte Input[22]
//     PlcTask Outputs/UN01.inf_EM07_M1.out/data @bit 184 <-> API/Term 2 (Modular)/EM07-M1/Outputs/1 Byte Input[23]
//     PlcTask Outputs/UN01.inf_EM07_M1.out/data @bit 192 <-> API/Term 2 (Modular)/EM07-M1/Outputs/1 Byte Input[24]
//     PlcTask Outputs/UN01.inf_EM07_M1.out/data @bit 200 <-> API/Term 2 (Modular)/EM07-M1/Outputs/1 Byte Input[25]
//     PlcTask Outputs/UN01.inf_EM07_M1.out/data @bit 208 <-> API/Term 2 (Modular)/EM07-M1/Outputs/1 Byte Input[26]
//     PlcTask Outputs/UN01.inf_EM07_M1.out/data @bit 216 <-> API/Term 2 (Modular)/EM07-M1/Outputs/1 Byte Input[27]
//     PlcTask Outputs/UN01.inf_EM07_M1.out/data @bit 224 <-> API/Term 2 (Modular)/EM07-M1/Outputs/1 Byte Input[28]
//     PlcTask Outputs/UN01.inf_EM07_M1.out/data @bit 232 <-> API/Term 2 (Modular)/EM07-M1/Outputs/1 Byte Input[29]
//     PlcTask Outputs/UN01.inf_EM07_M1.out/data @bit 16 <-> API/Term 2 (Modular)/EM07-M1/Outputs/1 Byte Input[2]
//     PlcTask Outputs/UN01.inf_EM07_M1.out/data @bit 240 <-> API/Term 2 (Modular)/EM07-M1/Outputs/1 Byte Input[30]
//     PlcTask Outputs/UN01.inf_EM07_M1.out/data @bit 248 <-> API/Term 2 (Modular)/EM07-M1/Outputs/1 Byte Input[31]
//     PlcTask Outputs/UN01.inf_EM07_M1.out/data @bit 24 <-> API/Term 2 (Modular)/EM07-M1/Outputs/1 Byte Input[3]
//     PlcTask Outputs/UN01.inf_EM07_M1.out/data @bit 32 <-> API/Term 2 (Modular)/EM07-M1/Outputs/1 Byte Input[4]
//     PlcTask Outputs/UN01.inf_EM07_M1.out/data @bit 40 <-> API/Term 2 (Modular)/EM07-M1/Outputs/1 Byte Input[5]
//     PlcTask Outputs/UN01.inf_EM07_M1.out/data @bit 48 <-> API/Term 2 (Modular)/EM07-M1/Outputs/1 Byte Input[6]
//     PlcTask Outputs/UN01.inf_EM07_M1.out/data @bit 56 <-> API/Term 2 (Modular)/EM07-M1/Outputs/1 Byte Input[7]
//     PlcTask Outputs/UN01.inf_EM07_M1.out/data @bit 64 <-> API/Term 2 (Modular)/EM07-M1/Outputs/1 Byte Input[8]
//     PlcTask Outputs/UN01.inf_EM07_M1.out/data @bit 72 <-> API/Term 2 (Modular)/EM07-M1/Outputs/1 Byte Input[9]
//     PlcTask Outputs/UN01.inf_EM08_M1.out/data @bit 80 <-> API/Term 2 (Modular)/EM08-M1/Outputs/1 Byte Input[10]
//     PlcTask Outputs/UN01.inf_EM08_M1.out/data @bit 88 <-> API/Term 2 (Modular)/EM08-M1/Outputs/1 Byte Input[11]
//     PlcTask Outputs/UN01.inf_EM08_M1.out/data @bit 96 <-> API/Term 2 (Modular)/EM08-M1/Outputs/1 Byte Input[12]
//     PlcTask Outputs/UN01.inf_EM08_M1.out/data @bit 104 <-> API/Term 2 (Modular)/EM08-M1/Outputs/1 Byte Input[13]
//     PlcTask Outputs/UN01.inf_EM08_M1.out/data @bit 112 <-> API/Term 2 (Modular)/EM08-M1/Outputs/1 Byte Input[14]
//     PlcTask Outputs/UN01.inf_EM08_M1.out/data @bit 120 <-> API/Term 2 (Modular)/EM08-M1/Outputs/1 Byte Input[15]
//     PlcTask Outputs/UN01.inf_EM08_M1.out/data @bit 128 <-> API/Term 2 (Modular)/EM08-M1/Outputs/1 Byte Input[16]
//     PlcTask Outputs/UN01.inf_EM08_M1.out/data @bit 136 <-> API/Term 2 (Modular)/EM08-M1/Outputs/1 Byte Input[17]
//     PlcTask Outputs/UN01.inf_EM08_M1.out/data @bit 144 <-> API/Term 2 (Modular)/EM08-M1/Outputs/1 Byte Input[18]
//     PlcTask Outputs/UN01.inf_EM08_M1.out/data @bit 152 <-> API/Term 2 (Modular)/EM08-M1/Outputs/1 Byte Input[19]
//     PlcTask Outputs/UN01.inf_EM08_M1.out/data @bit 8 <-> API/Term 2 (Modular)/EM08-M1/Outputs/1 Byte Input[1]
//     PlcTask Outputs/UN01.inf_EM08_M1.out/data @bit 160 <-> API/Term 2 (Modular)/EM08-M1/Outputs/1 Byte Input[20]
//     PlcTask Outputs/UN01.inf_EM08_M1.out/data @bit 168 <-> API/Term 2 (Modular)/EM08-M1/Outputs/1 Byte Input[21]
//     PlcTask Outputs/UN01.inf_EM08_M1.out/data @bit 176 <-> API/Term 2 (Modular)/EM08-M1/Outputs/1 Byte Input[22]
//     PlcTask Outputs/UN01.inf_EM08_M1.out/data @bit 184 <-> API/Term 2 (Modular)/EM08-M1/Outputs/1 Byte Input[23]
//     PlcTask Outputs/UN01.inf_EM08_M1.out/data @bit 192 <-> API/Term 2 (Modular)/EM08-M1/Outputs/1 Byte Input[24]
//     PlcTask Outputs/UN01.inf_EM08_M1.out/data @bit 200 <-> API/Term 2 (Modular)/EM08-M1/Outputs/1 Byte Input[25]
//     PlcTask Outputs/UN01.inf_EM08_M1.out/data @bit 208 <-> API/Term 2 (Modular)/EM08-M1/Outputs/1 Byte Input[26]
//     PlcTask Outputs/UN01.inf_EM08_M1.out/data @bit 216 <-> API/Term 2 (Modular)/EM08-M1/Outputs/1 Byte Input[27]
//     PlcTask Outputs/UN01.inf_EM08_M1.out/data @bit 224 <-> API/Term 2 (Modular)/EM08-M1/Outputs/1 Byte Input[28]
//     PlcTask Outputs/UN01.inf_EM08_M1.out/data @bit 232 <-> API/Term 2 (Modular)/EM08-M1/Outputs/1 Byte Input[29]
//     PlcTask Outputs/UN01.inf_EM08_M1.out/data @bit 16 <-> API/Term 2 (Modular)/EM08-M1/Outputs/1 Byte Input[2]
//     PlcTask Outputs/UN01.inf_EM08_M1.out/data @bit 240 <-> API/Term 2 (Modular)/EM08-M1/Outputs/1 Byte Input[30]
//     PlcTask Outputs/UN01.inf_EM08_M1.out/data @bit 248 <-> API/Term 2 (Modular)/EM08-M1/Outputs/1 Byte Input[31]
//     PlcTask Outputs/UN01.inf_EM08_M1.out/data @bit 24 <-> API/Term 2 (Modular)/EM08-M1/Outputs/1 Byte Input[3]
//     PlcTask Outputs/UN01.inf_EM08_M1.out/data @bit 32 <-> API/Term 2 (Modular)/EM08-M1/Outputs/1 Byte Input[4]
//     PlcTask Outputs/UN01.inf_EM08_M1.out/data @bit 40 <-> API/Term 2 (Modular)/EM08-M1/Outputs/1 Byte Input[5]
//     PlcTask Outputs/UN01.inf_EM08_M1.out/data @bit 48 <-> API/Term 2 (Modular)/EM08-M1/Outputs/1 Byte Input[6]
//     PlcTask Outputs/UN01.inf_EM08_M1.out/data @bit 56 <-> API/Term 2 (Modular)/EM08-M1/Outputs/1 Byte Input[7]
//     PlcTask Outputs/UN01.inf_EM08_M1.out/data @bit 64 <-> API/Term 2 (Modular)/EM08-M1/Outputs/1 Byte Input[8]
//     PlcTask Outputs/UN01.inf_EM08_M1.out/data @bit 72 <-> API/Term 2 (Modular)/EM08-M1/Outputs/1 Byte Input[9]
//   PLC1/PLC1 Instance <-> Device 4 (EtherCAT)
//     PlcTask Inputs/DeviceState.nDev4_DevState <-> Inputs/DevState
//   PLC1/PLC1 Instance <-> NC-Task 1 SAF/Axes/EM04-M1
//     PlcTask Inputs/UN01.EM04_M1.axis.NcToPlc <-> Outputs/ToPlc
//     PlcTask Outputs/UN01.EM04_M1.axis.PlcToNc <-> Inputs/FromPlc
//   PLC1/PLC1 Instance <-> NC-Task 1 SAF/Axes/EM05-M1
//     PlcTask Inputs/UN01.EM05_M1.axis.NcToPlc <-> Outputs/ToPlc
//     PlcTask Outputs/UN01.EM05_M1.axis.PlcToNc <-> Inputs/FromPlc
//   PLC1/PLC1 Instance <-> NC-Task 1 SAF/Axes/EM07-M1
//     PlcTask Inputs/UN01.EM07_M1.axis.NcToPlc <-> Outputs/ToPlc
//     PlcTask Outputs/UN01.EM07_M1.axis.PlcToNc <-> Inputs/FromPlc
//   PLC1/PLC1 Instance <-> NC-Task 1 SAF/Axes/EM08-M1
//     PlcTask Inputs/UN01.EM08_M1.axis.NcToPlc <-> Outputs/ToPlc
//     PlcTask Outputs/UN01.EM08_M1.axis.PlcToNc <-> Inputs/FromPlc

CONFIGURATION PLC1
    RESOURCE PLC ON TwinCAT3
        TASK PlcTask(INTERVAL := T#1ms, PRIORITY := 20);
        PROGRAM MAIN WITH PlcTask : MAIN;
    END_RESOURCE
END_CONFIGURATION

// ---- POUs/MAIN.TcPOU
PROGRAM MAIN
VAR
	nCounter	: INT;
END_VAR

nCounter:=nCounter+1;
UN01();
DeviceState();

END_PROGRAM

// ---- POUs/UN01.TcPOU
PROGRAM UN01
VAR
	EM04_M1 : SG_Servo.FB_EL72XX;
	inf_EM04_M1 : SG_Servo.FB_ItfServo;
	EM05_M1 : SG_Servo.FB_EL72XX;
	inf_EM05_M1 : SG_Servo.FB_ItfServo;
	EM07_M1 : SG_Servo.FB_EL72XX;
	inf_EM07_M1 : SG_Servo.FB_ItfServo;
	EM08_M1 : SG_Servo.FB_EL72XX;
	inf_EM08_M1 : SG_Servo.FB_ItfServo;
END_VAR

//EM04 Pallet conveyor
inf_EM04_M1.servo := EM04_M1;
inf_EM04_M1();
//EM05 Pallet conveyor
inf_EM05_M1.servo := EM05_M1;
inf_EM05_M1();
//EM07 Tub transfer
inf_EM07_M1.servo := EM07_M1;
inf_EM07_M1();
//EM08 Tub transfer in
inf_EM08_M1.servo := EM08_M1;
inf_EM08_M1();

END_PROGRAM

// ---- POUs/DeviceState.TcPOU
PROGRAM DeviceState
VAR
	nDev1_DevState AT %I* : UINT;
	nDev4_DevState AT %I* : UINT;
	nProfinetState AT %I* : UINT;
	nPnIoBoxState AT %I* : UINT;
	nPnIoBoxCtrl AT %Q* : UINT;
	nState		: UINT;
	bReset		: BOOL;
	bErrorBit	: BOOL;
	tDelay		: TON;
	tPulse		: TON;
END_VAR

;
(*
bErrorBit		:= nPnIoBoxState.3;
nPnIoBoxCtrl.0	:= bReset;

CASE nState OF
	
	0:
	IF nProfinetState <> 8 OR bErrorBit THEN
		tDelay(IN:=TRUE , PT:=T#5S);
		IF tDelay.Q THEN
			tPulse(IN:=TRUE , PT:=T#1S);
			bReset	:= TRUE;
			nState	:= 10;
		END_IF
	ELSE
		tDelay(IN:=FALSE);	
	END_IF
	
	10:
	tPulse();
	IF tPulse.Q THEN
		bReset	:= FALSE;
		tDelay(IN:=FALSE);
		tPulse(IN:=FALSE);
		nState	:= 0;	
	END_IF
	
END_CASE
*)

END_PROGRAM
